PROGRAM MAIN
VAR
	Belt1Start					:	BOOL;
	Belt2Start					:	BOOL;
	Belt1Stop					:	BOOL;
	Belt2Stop					:	BOOL;
	Belt1Guard					:	BOOL;
	Belt2Guard					:	BOOL;
	Belt3Guard					:	BOOL;
	
	srBelt1LampOn				:	SR;
	srBelt2LampOn				:	SR;
	Belt1LampOn					:	BOOL;
	Belt2LampOn					:	BOOL;
	Belt1LampOff				:	BOOL;
	Belt2LampOff				:	BOOL;
	
	MotorBelt1					:	BOOL;
	MotorBelt2					:	BOOL;
	MotorBelt3					:	BOOL;
	
	Pulse2Hz					:	BOOL;
	
	tonStartPhase				:	TON;
	tonBelt12MonitorTime		:	TON;
	tonBelt3MonitorTime			:	TON;
	tofDelayOffBelt1			:	TOF;
	tofDelayOffBelt2			:	TOF;
	tofDelayOffBelt3			:	TOF;
	
	tpBlink01					: TP;
	tpBlink02					: TP;
END_VAR

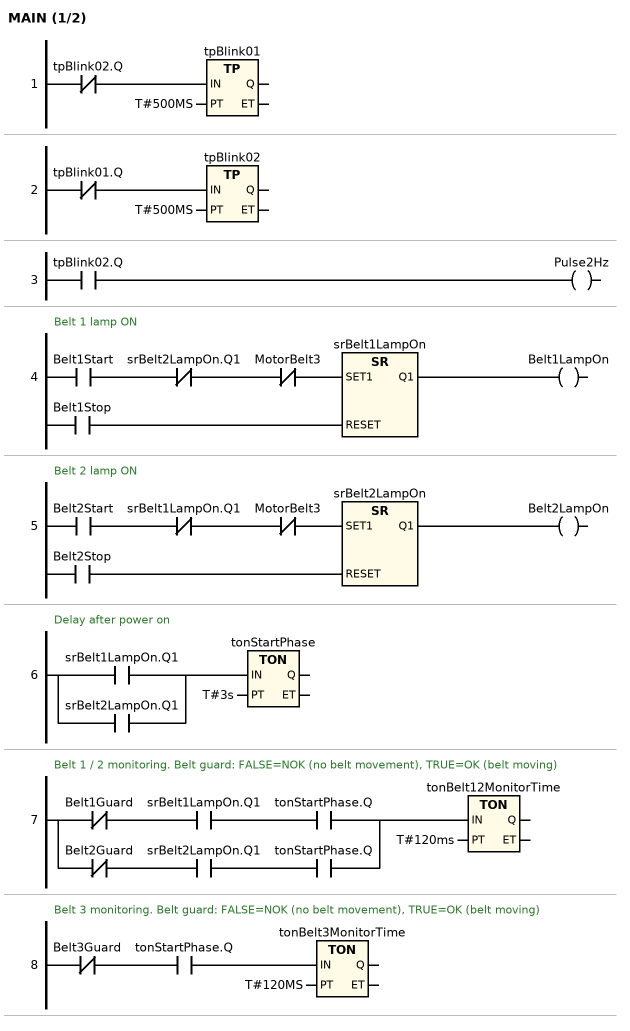
// NETWORK 1
tpBlink01(IN := NOT tpBlink02.Q, PT := T#500MS); // TP

// NETWORK 2
tpBlink02(IN := NOT tpBlink01.Q, PT := T#500MS); // TP

// NETWORK 3
Pulse2Hz := tpBlink02.Q;

// NETWORK 4
// Belt 1 lamp ON
srBelt1LampOn(SET1 := Belt1Start AND NOT srBelt2LampOn.Q1 AND NOT MotorBelt3, RESET := Belt1Stop); // SR
Belt1LampOn := srBelt1LampOn.Q1;

// NETWORK 5
// Belt 2 lamp ON
srBelt2LampOn(SET1 := Belt2Start AND NOT srBelt1LampOn.Q1 AND NOT MotorBelt3, RESET := Belt2Stop); // SR
Belt2LampOn := srBelt2LampOn.Q1;

// NETWORK 6
// Delay after power on
tonStartPhase(IN := srBelt1LampOn.Q1 OR srBelt2LampOn.Q1, PT := T#3s); // TON

// NETWORK 7
// Belt 1 / 2 monitoring. Belt guard: FALSE=NOK (no belt movement), TRUE=OK (belt moving)
tonBelt12MonitorTime(IN := NOT Belt1Guard AND srBelt1LampOn.Q1 AND tonStartPhase.Q OR NOT Belt2Guard AND srBelt2LampOn.Q1 AND tonStartPhase.Q, PT := T#120ms); // TON

// NETWORK 8
// Belt 3 monitoring. Belt guard: FALSE=NOK (no belt movement), TRUE=OK (belt moving)
tonBelt3MonitorTime(IN := NOT Belt3Guard AND tonStartPhase.Q, PT := T#120MS); // TON

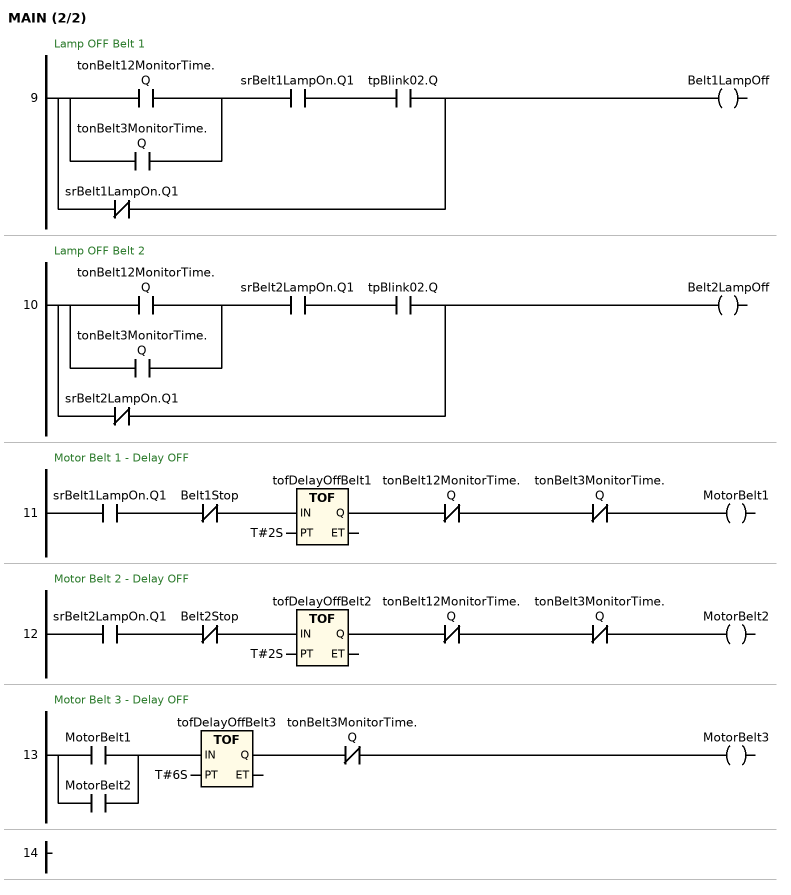
// NETWORK 9
// Lamp OFF Belt 1
Belt1LampOff := (tonBelt12MonitorTime.Q OR tonBelt3MonitorTime.Q) AND srBelt1LampOn.Q1 AND tpBlink02.Q OR NOT srBelt1LampOn.Q1;

// NETWORK 10
// Lamp OFF Belt 2
Belt2LampOff := (tonBelt12MonitorTime.Q OR tonBelt3MonitorTime.Q) AND srBelt2LampOn.Q1 AND tpBlink02.Q OR NOT srBelt2LampOn.Q1;

// NETWORK 11
// Motor Belt 1 - Delay OFF
tofDelayOffBelt1(IN := srBelt1LampOn.Q1 AND NOT Belt1Stop, PT := T#2S); // TOF
MotorBelt1 := tofDelayOffBelt1.Q AND NOT tonBelt12MonitorTime.Q AND NOT tonBelt3MonitorTime.Q;

// NETWORK 12
// Motor Belt 2 - Delay OFF
tofDelayOffBelt2(IN := srBelt2LampOn.Q1 AND NOT Belt2Stop, PT := T#2S); // TOF
MotorBelt2 := tofDelayOffBelt2.Q AND NOT tonBelt12MonitorTime.Q AND NOT tonBelt3MonitorTime.Q;

// NETWORK 13
// Motor Belt 3 - Delay OFF
tofDelayOffBelt3(IN := MotorBelt1 OR MotorBelt2, PT := T#6S); // TOF
MotorBelt3 := tofDelayOffBelt3.Q AND NOT tonBelt3MonitorTime.Q;

// NETWORK 14

END_PROGRAM

(* stored: Version 1.1.0.1, ProductVersion 3.1.4024.15
   POU MAIN: Id {f61e646b-8cdf-4734-bb25-59a0dba1df8e}, SpecialFunc None *)
